(* IEC 61131-3 sources: CodesysTest/export/Function Blocks/SolenoidValves/FB_PneumaticActuator.pou, 1 file *)

(* ---- FB_PneumaticActuator.pou.st ---- *)
(*#-#-#-#-#-#-#-#-#-#---Declaration---#-#-#-#-#-#-#-#-#-#-#-#-#*)

FUNCTION_BLOCK FB_PneumaticActuator EXTENDS FB_SolenoidValve IMPLEMENTS ICylinder
VAR_INPUT
END_VAR
VAR_OUTPUT
END_VAR
VAR
	_extendAsserted : BOOL;
	_isExtended : BOOL;
	_retractAsserted : BOOL;
	_isRetracted : BOOL;
END_VAR
(*#-#-#-#-#-#-#-#-#-#---Implementation---#-#-#-#-#-#-#-#-#-#-#-#-#*)
